{attribute 'GeneratedUsingTerminal: EP7402-0057-0017'}
{attribute addProperty BoxType "EP7402-0057-0017"}
{attribute addProperty Id "DI_InputsAT %I*DI_Inputs_58955D1A8STM_Status_Channel_1AT %I*STM_Status_Channel_99D1DFFA7STM_Synchron_info_data_Channel_1AT %I*STM_Synchron_info_data_Channel_DD535D916STM_Status_Channel_2AT %I*STM_Status_Channel_99D1DFFA7STM_Synchron_info_data_Channel_2AT %I*STM_Synchron_info_data_Channel_DD535D916STM_Inputs_DeviceAT %I*STM_Inputs_Device_A41D845621DO_OutputsAT %Q*DO_Outputs_A241BD3A8STM_Control_Channel_1AT %Q*STM_Control_Channel_F193EBCD4STM_Target_Velocity_Channel_1AT %Q*STM_Target_Velocity_Channel_E69D83256STM_Control_Channel_2AT %Q*STM_Control_Channel_F193EBCD4STM_Target_Velocity_Channel_2AT %Q*STM_Target_Velocity_Channel_E69D83256WcStateAT %I*WcState_9091E0EB2InfoDataAT %I*InfoData_F796F5796"}
{attribute addProperty CRC "2823262412"}
{attribute addProperty Size "91"}
TYPE EP7402_A84790CC EXTENDS EtcSlaveTerminalBase_947E5A46 :
STRUCT
	{attribute addProperty Name "DI_Inputs"}
	DI_Inputs : DI_Inputs_58955D1A;
	{attribute addProperty Name "STM_Status_Channel_1"}
	STM_Status_Channel_1 : STM_Status_Channel_99D1DFFA;
	{attribute addProperty Name "STM_Synchron_info_data_Channel_1"}
	STM_Synchron_info_data_Channel_1 : STM_Synchron_info_data_Channel_DD535D91;
	{attribute addProperty Name "STM_Status_Channel_2"}
	STM_Status_Channel_2 : STM_Status_Channel_99D1DFFA;
	{attribute addProperty Name "STM_Synchron_info_data_Channel_2"}
	STM_Synchron_info_data_Channel_2 : STM_Synchron_info_data_Channel_DD535D91;
	{attribute addProperty Name "STM_Inputs_Device"}
	STM_Inputs_Device : STM_Inputs_Device_A41D8456;
	{attribute addProperty Name "DO_Outputs"}
	DO_Outputs : DO_Outputs_A241BD3A;
	{attribute addProperty Name "STM_Control_Channel_1"}
	STM_Control_Channel_1 : STM_Control_Channel_F193EBCD;
	{attribute addProperty Name "STM_Target_Velocity_Channel_1"}
	STM_Target_Velocity_Channel_1 : STM_Target_Velocity_Channel_E69D8325;
	{attribute addProperty Name "STM_Control_Channel_2"}
	STM_Control_Channel_2 : STM_Control_Channel_F193EBCD;
	{attribute addProperty Name "STM_Target_Velocity_Channel_2"}
	STM_Target_Velocity_Channel_2 : STM_Target_Velocity_Channel_E69D8325;
	{attribute addProperty Name "WcState"}
	WcState : WcState_9091E0EB;
	{attribute addProperty Name "InfoData"}
	InfoData : InfoData_F796F579;
END_STRUCT
END_TYPE

(* stored: Version 1.2.0.0, ProductVersion 3.1.4024.9
   DUT EP7402_A84790CC: Id {1ce330b8-c1ae-48a6-9b50-0b4fe0360685} *)
